{attribute 'GeneratedUsingTerminal: EK1100-0000-0018'}
{attribute addProperty BoxType "EK1100-0000-0018"}
{attribute addProperty Id "Beckhoff_EPP3xxxEK1122Beckhoff_EPP3xxxEK1122_A76E71A71480"}
{attribute addProperty CRC "939452576"}
{attribute addProperty Size "1480"}
TYPE Beckhoff_EPP3xxx_37FEE8A0 EXTENDS EK1100_1FC0878B :
STRUCT
	{attribute addProperty Name "Beckhoff EPP3xxxEK1122"}
	{attribute addProperty PreviousPort "Beckhoff EPP3xxx : B"}
	Beckhoff_EPP3xxxEK1122 : Beckhoff_EPP3xxxEK1122_A76E71A7;
END_STRUCT
END_TYPE

(* stored: Version 1.2.0.0, ProductVersion 3.1.4024.9
   DUT Beckhoff_EPP3xxx_37FEE8A0: Id {78c45621-c0bf-47a5-87c8-0dc20ee502be} *)
